{attribute addProperty BoxType "EK1122-0000-0018"}
{attribute addProperty Id "Beckhoff_EPP5xxxsub_EK1100EK1100_179A0949162A_0001_EPP5001_0002_0016EPP5001_636E7B5014418A_0002_EPP5101_0002_0016EPP5101_F338D8E417622A_0003_EPP5101_0002_0017EPP5101_F338D8E417622A_0004_EPP5101_0011_0016EPP5101_BA9EF92517622A_0005_EPP5101_0011_0017EPP5101_BA9EF92517622A_0006_EPP5101_1002_0016EPP5101_F338D8E417622A_0007_EPP5101_1002_0017EPP5101_F338D8E417622A_0008_EPP5151_0002_0016EPP5151_BA9EF92517622A_0009_EPP5151_0002_0017EPP5151_BA9EF92517622"}
{attribute addProperty CRC "2752445838"}
{attribute addProperty SizeInBites "1568"}
{attribute addProperty SizeInBytes "196"}
TYPE Beckhoff_EPP5xxxEK1122_A40EFD8E EXTENDS EK1122_179A0949 :
STRUCT
	{attribute addProperty Name "Beckhoff_EPP5xxxsub_EK1100"}
	Beckhoff_EPP5xxxsub_EK1100 : EK1100_179A0949;
	{attribute addProperty Name "A_0001_EPP5001_0002_0016"}
	A_0001_EPP5001_0002_0016 : EPP5001_636E7B50;
	{attribute addProperty Name "A_0002_EPP5101_0002_0016"}
	A_0002_EPP5101_0002_0016 : EPP5101_F338D8E4;
	{attribute addProperty Name "A_0003_EPP5101_0002_0017"}
	A_0003_EPP5101_0002_0017 : EPP5101_F338D8E4;
	{attribute addProperty Name "A_0004_EPP5101_0011_0016"}
	A_0004_EPP5101_0011_0016 : EPP5101_BA9EF925;
	{attribute addProperty Name "A_0005_EPP5101_0011_0017"}
	A_0005_EPP5101_0011_0017 : EPP5101_BA9EF925;
	{attribute addProperty Name "A_0006_EPP5101_1002_0016"}
	A_0006_EPP5101_1002_0016 : EPP5101_F338D8E4;
	{attribute addProperty Name "A_0007_EPP5101_1002_0017"}
	A_0007_EPP5101_1002_0017 : EPP5101_F338D8E4;
	{attribute addProperty Name "A_0008_EPP5151_0002_0016"}
	A_0008_EPP5151_0002_0016 : EPP5151_BA9EF925;
	{attribute addProperty Name "A_0009_EPP5151_0002_0017"}
	A_0009_EPP5151_0002_0017 : EPP5151_BA9EF925;
END_STRUCT
END_TYPE

(* stored: Version 1.2.0.0, ProductVersion 3.1.4024.9
   DUT Beckhoff_EPP5xxxEK1122_A40EFD8E: Id {f93f9faa-e5b4-419d-850b-e47c71ea165d} *)
